// Since FB_ErrorSource is an ABSTRACT class, the functionality needs to be implemented by extending the base class
FUNCTION_BLOCK INTERNAL FB_ErrorSource_ExtensionForTests EXTENDS FB_ErrorSource
VAR_INPUT
	eAdsErrorCodeToTest 	: TcError.AdsErrorCodes;
	sGenericErrorMessage	: Tc2_System.T_MaxString;
	nGenericErrorCode		: DINT;
	bError					: BOOL;		
END_VAR

THIS^.AdsError.Code := eAdsErrorCodeToTest;
THIS^.GenericError.Message := sGenericErrorMessage;
THIS^.GenericError.Code := nGenericErrorCode;
THIS^.Error := bError;

END_FUNCTION_BLOCK

(* stored: Version 1.1.0.1, ProductVersion 3.1.4024.14
   POU FB_ErrorSource_ExtensionForTests: Id {355c57f6-e53e-0e78-2d76-4f4befeabef0}, SpecialFunc None *)
